PROGRAM _1_LASER
VAR
	FB_LASER_SOURCE_MAXPHOTONICS1: FB_LASER_SOURCE_MAXPHOTONICS;
	FB_LASER_TETE_RAYTOOLS1: FB_LASER_TETE_RAYTOOLS_1;

	Dem_Serrage_Presseur_Entree: BOOL;
	Dem_Desserrage_Presseur_Entree: BOOL;
	Pos_Reelle_Presseur_Entree_D: LREAL;
	Pos_Reelle_Presseur_Entree_G: LREAL;

	Dem_Serrage_Presseur_Sortie: BOOL;
	Dem_Desserrage_Presseur_Sortie: BOOL;
	Pos_Reelle_Presseur_Sortie_D: LREAL;
	Pos_Reelle_Presseur_Sortie_G: LREAL;


	Div_Zero: BOOL;

	Chgt_Plan_Aile_Ref: FB_Calcul_Chgt_Origine_Plan;
	Chgt_Plan_Ame: FB_Calcul_Chgt_Origine_Plan;
	Chgt_Plan_Aile_Opp_Ref: FB_Calcul_Chgt_Origine_Plan;
	
	Feedback_Laser_Power: USINT;
	Feedback_Laser_Duty: USINT;
	Feedback_Laser_Freq: UINT;
	Feedback_Laser_Power_Watts	:UDINT;
	
	
	MeS_Aspiration	:TOF;
	Test_aspi: BOOL;
	Refroidissement	:TOF;
	Test_Refroidissement	:BOOL;
END_VAR
VAR // added by the converter: edge detectors and wires of the graphical bodies
    _w1 : BOOL;
END_VAR

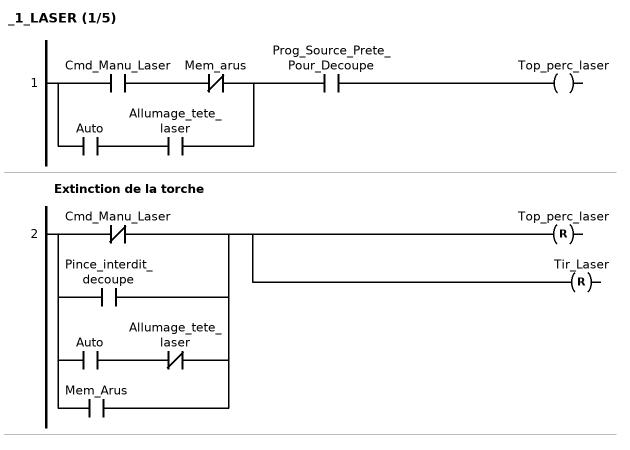
// NETWORK 1
Top_perc_laser := (Cmd_Manu_Laser AND NOT Mem_arus OR Auto AND Allumage_tete_laser) AND Prog_Source_Prete_Pour_Decoupe;

// NETWORK 2: Extinction de la torche
_w1 := NOT Cmd_Manu_Laser OR Pince_interdit_decoupe OR Auto AND NOT Allumage_tete_laser OR Mem_Arus;
Top_perc_laser R= _w1;
Tir_Laser R= _w1;

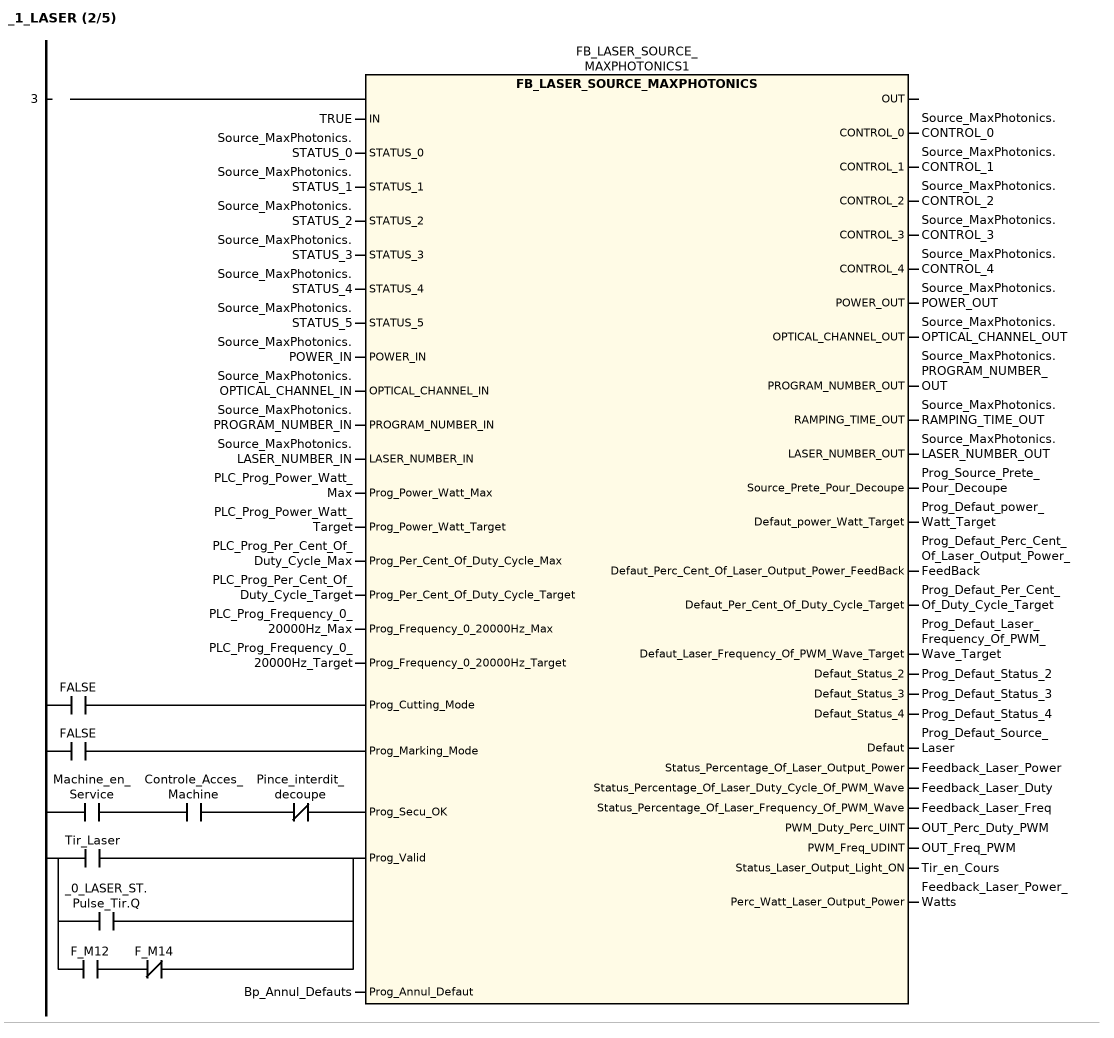
// NETWORK 3
FB_LASER_SOURCE_MAXPHOTONICS1(
    IN := TRUE,
    STATUS_0 := Source_MaxPhotonics.STATUS_0,
    STATUS_1 := Source_MaxPhotonics.STATUS_1,
    STATUS_2 := Source_MaxPhotonics.STATUS_2,
    STATUS_3 := Source_MaxPhotonics.STATUS_3,
    STATUS_4 := Source_MaxPhotonics.STATUS_4,
    STATUS_5 := Source_MaxPhotonics.STATUS_5,
    POWER_IN := Source_MaxPhotonics.POWER_IN,
    OPTICAL_CHANNEL_IN := Source_MaxPhotonics.OPTICAL_CHANNEL_IN,
    PROGRAM_NUMBER_IN := Source_MaxPhotonics.PROGRAM_NUMBER_IN,
    LASER_NUMBER_IN := Source_MaxPhotonics.LASER_NUMBER_IN,
    Prog_Power_Watt_Max := PLC_Prog_Power_Watt_Max,
    Prog_Power_Watt_Target := PLC_Prog_Power_Watt_Target,
    Prog_Per_Cent_Of_Duty_Cycle_Max := PLC_Prog_Per_Cent_Of_Duty_Cycle_Max,
    Prog_Per_Cent_Of_Duty_Cycle_Target := PLC_Prog_Per_Cent_Of_Duty_Cycle_Target,
    Prog_Frequency_0_20000Hz_Max := PLC_Prog_Frequency_0_20000Hz_Max,
    Prog_Frequency_0_20000Hz_Target := PLC_Prog_Frequency_0_20000Hz_Target,
    Prog_Cutting_Mode := FALSE,
    Prog_Marking_Mode := FALSE,
    Prog_Secu_OK := Machine_en_Service AND Controle_Acces_Machine AND NOT Pince_interdit_decoupe,
    Prog_Valid := Tir_Laser OR _0_LASER_ST.Pulse_Tir.Q OR F_M12 AND NOT F_M14,
    Prog_Annul_Defaut := Bp_Annul_Defauts,
    CONTROL_0 => Source_MaxPhotonics.CONTROL_0,
    CONTROL_1 => Source_MaxPhotonics.CONTROL_1,
    CONTROL_2 => Source_MaxPhotonics.CONTROL_2,
    CONTROL_3 => Source_MaxPhotonics.CONTROL_3,
    CONTROL_4 => Source_MaxPhotonics.CONTROL_4,
    POWER_OUT => Source_MaxPhotonics.POWER_OUT,
    OPTICAL_CHANNEL_OUT => Source_MaxPhotonics.OPTICAL_CHANNEL_OUT,
    PROGRAM_NUMBER_OUT => Source_MaxPhotonics.PROGRAM_NUMBER_OUT,
    RAMPING_TIME_OUT => Source_MaxPhotonics.RAMPING_TIME_OUT,
    LASER_NUMBER_OUT => Source_MaxPhotonics.LASER_NUMBER_OUT,
    Source_Prete_Pour_Decoupe => Prog_Source_Prete_Pour_Decoupe,
    Defaut_power_Watt_Target => Prog_Defaut_power_Watt_Target,
    Defaut_Perc_Cent_Of_Laser_Output_Power_FeedBack => Prog_Defaut_Perc_Cent_Of_Laser_Output_Power_FeedBack,
    Defaut_Per_Cent_Of_Duty_Cycle_Target => Prog_Defaut_Per_Cent_Of_Duty_Cycle_Target,
    Defaut_Laser_Frequency_Of_PWM_Wave_Target => Prog_Defaut_Laser_Frequency_Of_PWM_Wave_Target,
    Defaut_Status_2 => Prog_Defaut_Status_2,
    Defaut_Status_3 => Prog_Defaut_Status_3,
    Defaut_Status_4 => Prog_Defaut_Status_4,
    Defaut => Prog_Defaut_Source_Laser,
    Status_Percentage_Of_Laser_Output_Power => Feedback_Laser_Power,
    Status_Percentage_Of_Laser_Duty_Cycle_Of_PWM_Wave => Feedback_Laser_Duty,
    Status_Percentage_Of_Laser_Frequency_Of_PWM_Wave => Feedback_Laser_Freq,
    PWM_Duty_Perc_UINT => OUT_Perc_Duty_PWM,
    PWM_Freq_UDINT => OUT_Freq_PWM,
    Status_Laser_Output_Light_ON => Tir_en_Cours,
    Perc_Watt_Laser_Output_Power => Feedback_Laser_Power_Watts); // FB_LASER_SOURCE_MAXPHOTONICS

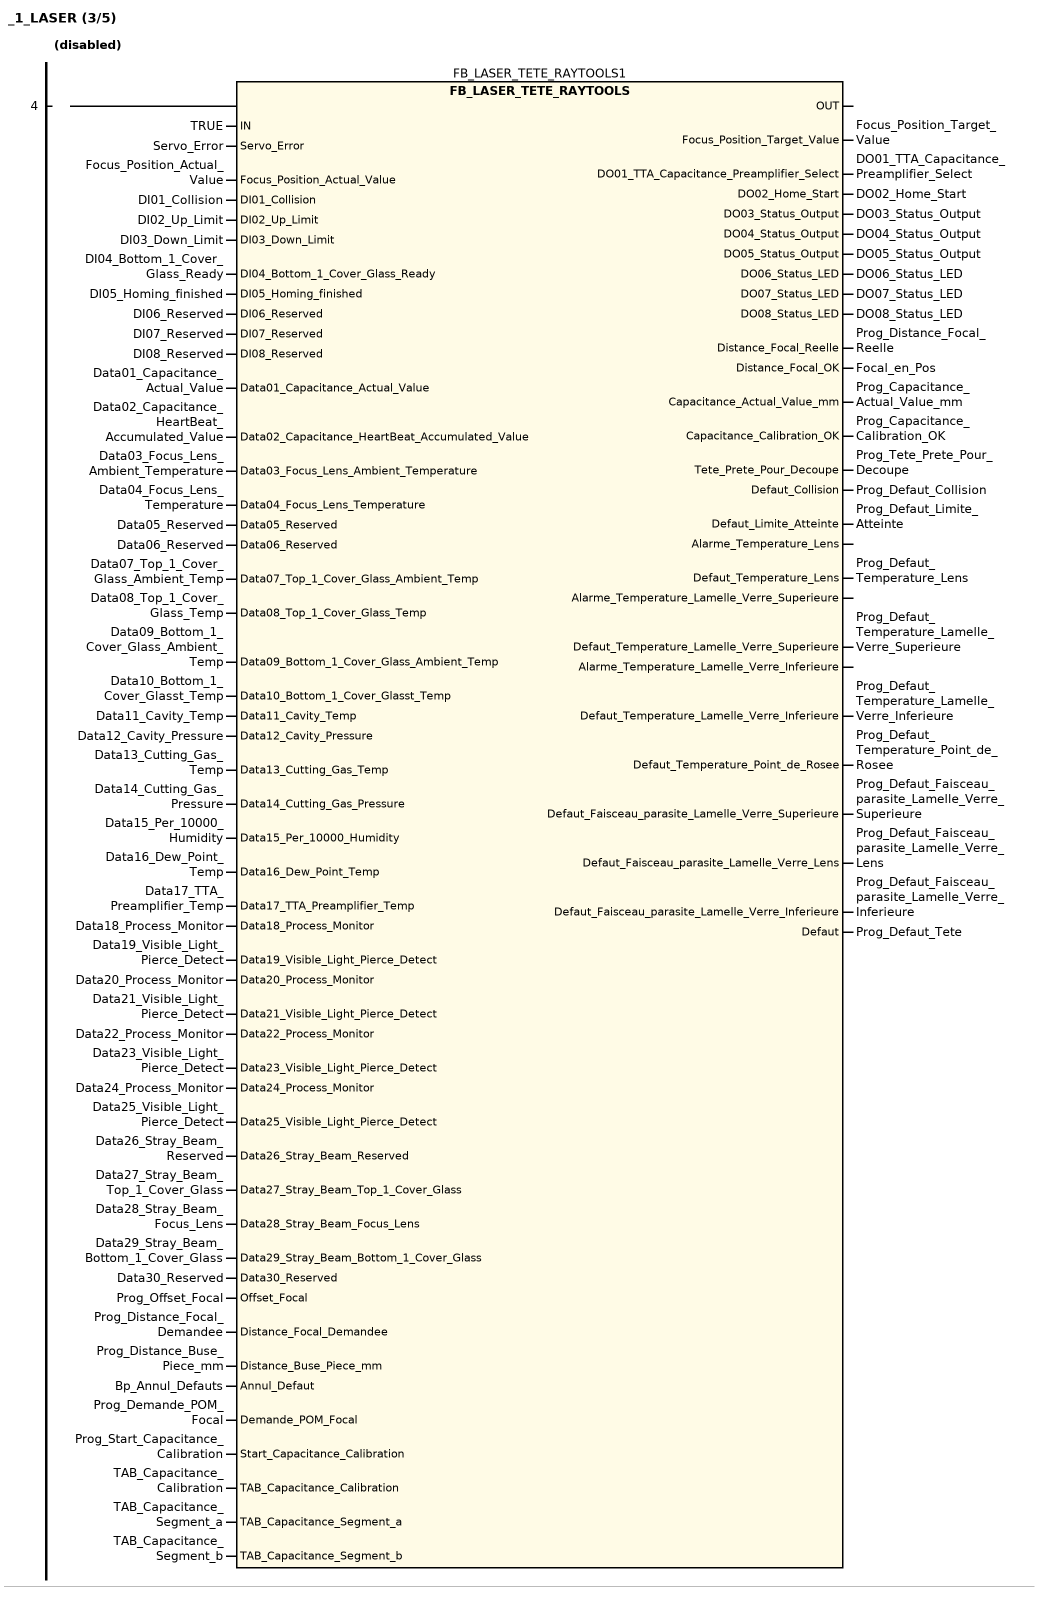
// NETWORK 4 (disabled)
// FB_LASER_TETE_RAYTOOLS1(
//     IN := TRUE,
//     Servo_Error := Servo_Error,
//     Focus_Position_Actual_Value := Focus_Position_Actual_Value,
//     DI01_Collision := DI01_Collision,
//     DI02_Up_Limit := DI02_Up_Limit,
//     DI03_Down_Limit := DI03_Down_Limit,
//     DI04_Bottom_1_Cover_Glass_Ready := DI04_Bottom_1_Cover_Glass_Ready,
//     DI05_Homing_finished := DI05_Homing_finished,
//     DI06_Reserved := DI06_Reserved,
//     DI07_Reserved := DI07_Reserved,
//     DI08_Reserved := DI08_Reserved,
//     Data01_Capacitance_Actual_Value := Data01_Capacitance_Actual_Value,
//     Data02_Capacitance_HeartBeat_Accumulated_Value := Data02_Capacitance_HeartBeat_Accumulated_Value,
//     Data03_Focus_Lens_Ambient_Temperature := Data03_Focus_Lens_Ambient_Temperature,
//     Data04_Focus_Lens_Temperature := Data04_Focus_Lens_Temperature,
//     Data05_Reserved := Data05_Reserved,
//     Data06_Reserved := Data06_Reserved,
//     Data07_Top_1_Cover_Glass_Ambient_Temp := Data07_Top_1_Cover_Glass_Ambient_Temp,
//     Data08_Top_1_Cover_Glass_Temp := Data08_Top_1_Cover_Glass_Temp,
//     Data09_Bottom_1_Cover_Glass_Ambient_Temp := Data09_Bottom_1_Cover_Glass_Ambient_Temp,
//     Data10_Bottom_1_Cover_Glasst_Temp := Data10_Bottom_1_Cover_Glasst_Temp,
//     Data11_Cavity_Temp := Data11_Cavity_Temp,
//     Data12_Cavity_Pressure := Data12_Cavity_Pressure,
//     Data13_Cutting_Gas_Temp := Data13_Cutting_Gas_Temp,
//     Data14_Cutting_Gas_Pressure := Data14_Cutting_Gas_Pressure,
//     Data15_Per_10000_Humidity := Data15_Per_10000_Humidity,
//     Data16_Dew_Point_Temp := Data16_Dew_Point_Temp,
//     Data17_TTA_Preamplifier_Temp := Data17_TTA_Preamplifier_Temp,
//     Data18_Process_Monitor := Data18_Process_Monitor,
//     Data19_Visible_Light_Pierce_Detect := Data19_Visible_Light_Pierce_Detect,
//     Data20_Process_Monitor := Data20_Process_Monitor,
//     Data21_Visible_Light_Pierce_Detect := Data21_Visible_Light_Pierce_Detect,
//     Data22_Process_Monitor := Data22_Process_Monitor,
//     Data23_Visible_Light_Pierce_Detect := Data23_Visible_Light_Pierce_Detect,
//     Data24_Process_Monitor := Data24_Process_Monitor,
//     Data25_Visible_Light_Pierce_Detect := Data25_Visible_Light_Pierce_Detect,
//     Data26_Stray_Beam_Reserved := Data26_Stray_Beam_Reserved,
//     Data27_Stray_Beam_Top_1_Cover_Glass := Data27_Stray_Beam_Top_1_Cover_Glass,
//     Data28_Stray_Beam_Focus_Lens := Data28_Stray_Beam_Focus_Lens,
//     Data29_Stray_Beam_Bottom_1_Cover_Glass := Data29_Stray_Beam_Bottom_1_Cover_Glass,
//     Data30_Reserved := Data30_Reserved,
//     Offset_Focal := Prog_Offset_Focal,
//     Distance_Focal_Demandee := Prog_Distance_Focal_Demandee,
//     Distance_Buse_Piece_mm := Prog_Distance_Buse_Piece_mm,
//     Annul_Defaut := Bp_Annul_Defauts,
//     Demande_POM_Focal := Prog_Demande_POM_Focal,
//     Start_Capacitance_Calibration := Prog_Start_Capacitance_Calibration,
//     TAB_Capacitance_Calibration := TAB_Capacitance_Calibration,
//     TAB_Capacitance_Segment_a := TAB_Capacitance_Segment_a,
//     TAB_Capacitance_Segment_b := TAB_Capacitance_Segment_b,
//     Focus_Position_Target_Value => Focus_Position_Target_Value,
//     DO01_TTA_Capacitance_Preamplifier_Select => DO01_TTA_Capacitance_Preamplifier_Select,
//     DO02_Home_Start => DO02_Home_Start,
//     DO03_Status_Output => DO03_Status_Output,
//     DO04_Status_Output => DO04_Status_Output,
//     DO05_Status_Output => DO05_Status_Output,
//     DO06_Status_LED => DO06_Status_LED,
//     DO07_Status_LED => DO07_Status_LED,
//     DO08_Status_LED => DO08_Status_LED,
//     Distance_Focal_Reelle => Prog_Distance_Focal_Reelle,
//     Distance_Focal_OK => Focal_en_Pos,
//     Capacitance_Actual_Value_mm => Prog_Capacitance_Actual_Value_mm,
//     Capacitance_Calibration_OK => Prog_Capacitance_Calibration_OK,
//     Tete_Prete_Pour_Decoupe => Prog_Tete_Prete_Pour_Decoupe,
//     Defaut_Collision => Prog_Defaut_Collision,
//     Defaut_Limite_Atteinte => Prog_Defaut_Limite_Atteinte,
//     Defaut_Temperature_Lens => Prog_Defaut_Temperature_Lens,
//     Defaut_Temperature_Lamelle_Verre_Superieure => Prog_Defaut_Temperature_Lamelle_Verre_Superieure,
//     Defaut_Temperature_Lamelle_Verre_Inferieure => Prog_Defaut_Temperature_Lamelle_Verre_Inferieure,
//     Defaut_Temperature_Point_de_Rosee => Prog_Defaut_Temperature_Point_de_Rosee,
//     Defaut_Faisceau_parasite_Lamelle_Verre_Superieure => Prog_Defaut_Faisceau_parasite_Lamelle_Verre_Superieure,
//     Defaut_Faisceau_parasite_Lamelle_Verre_Lens => Prog_Defaut_Faisceau_parasite_Lamelle_Verre_Lens,
//     Defaut_Faisceau_parasite_Lamelle_Verre_Inferieure => Prog_Defaut_Faisceau_parasite_Lamelle_Verre_Inferieure,
//     Defaut => Prog_Defaut_Tete); // FB_LASER_TETE_RAYTOOLS

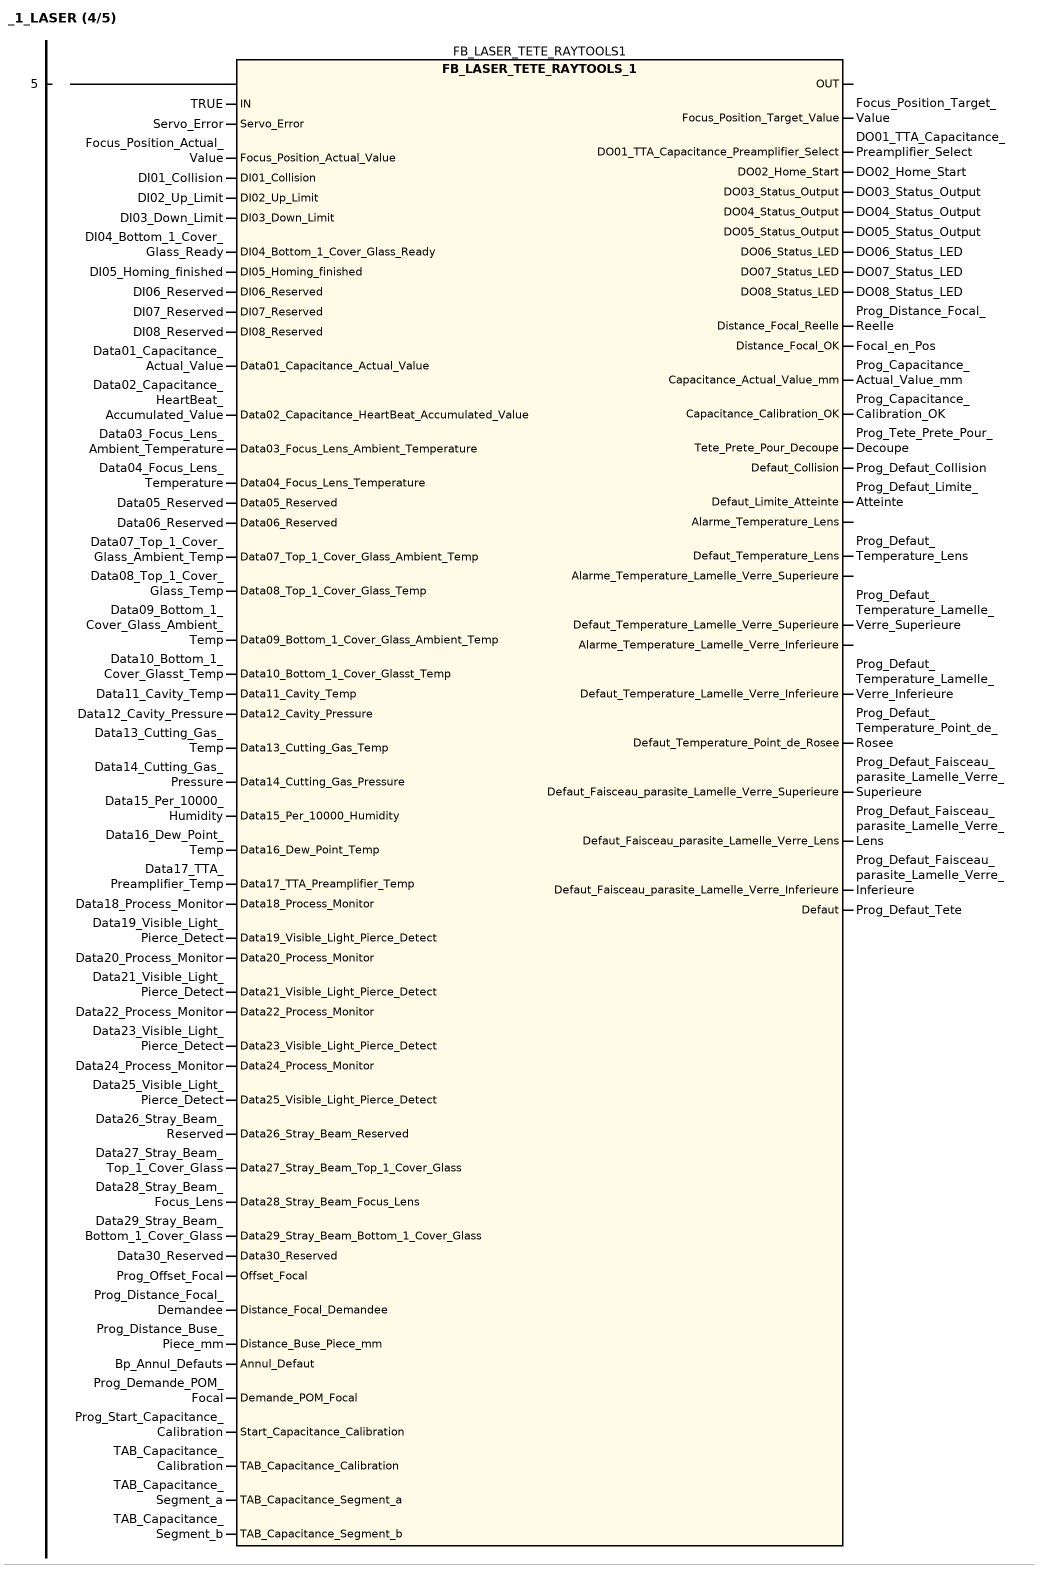
// NETWORK 5
FB_LASER_TETE_RAYTOOLS1(
    IN := TRUE,
    Servo_Error := Servo_Error,
    Focus_Position_Actual_Value := Focus_Position_Actual_Value,
    DI01_Collision := DI01_Collision,
    DI02_Up_Limit := DI02_Up_Limit,
    DI03_Down_Limit := DI03_Down_Limit,
    DI04_Bottom_1_Cover_Glass_Ready := DI04_Bottom_1_Cover_Glass_Ready,
    DI05_Homing_finished := DI05_Homing_finished,
    DI06_Reserved := DI06_Reserved,
    DI07_Reserved := DI07_Reserved,
    DI08_Reserved := DI08_Reserved,
    Data01_Capacitance_Actual_Value := Data01_Capacitance_Actual_Value,
    Data02_Capacitance_HeartBeat_Accumulated_Value := Data02_Capacitance_HeartBeat_Accumulated_Value,
    Data03_Focus_Lens_Ambient_Temperature := Data03_Focus_Lens_Ambient_Temperature,
    Data04_Focus_Lens_Temperature := Data04_Focus_Lens_Temperature,
    Data05_Reserved := Data05_Reserved,
    Data06_Reserved := Data06_Reserved,
    Data07_Top_1_Cover_Glass_Ambient_Temp := Data07_Top_1_Cover_Glass_Ambient_Temp,
    Data08_Top_1_Cover_Glass_Temp := Data08_Top_1_Cover_Glass_Temp,
    Data09_Bottom_1_Cover_Glass_Ambient_Temp := Data09_Bottom_1_Cover_Glass_Ambient_Temp,
    Data10_Bottom_1_Cover_Glasst_Temp := Data10_Bottom_1_Cover_Glasst_Temp,
    Data11_Cavity_Temp := Data11_Cavity_Temp,
    Data12_Cavity_Pressure := Data12_Cavity_Pressure,
    Data13_Cutting_Gas_Temp := Data13_Cutting_Gas_Temp,
    Data14_Cutting_Gas_Pressure := Data14_Cutting_Gas_Pressure,
    Data15_Per_10000_Humidity := Data15_Per_10000_Humidity,
    Data16_Dew_Point_Temp := Data16_Dew_Point_Temp,
    Data17_TTA_Preamplifier_Temp := Data17_TTA_Preamplifier_Temp,
    Data18_Process_Monitor := Data18_Process_Monitor,
    Data19_Visible_Light_Pierce_Detect := Data19_Visible_Light_Pierce_Detect,
    Data20_Process_Monitor := Data20_Process_Monitor,
    Data21_Visible_Light_Pierce_Detect := Data21_Visible_Light_Pierce_Detect,
    Data22_Process_Monitor := Data22_Process_Monitor,
    Data23_Visible_Light_Pierce_Detect := Data23_Visible_Light_Pierce_Detect,
    Data24_Process_Monitor := Data24_Process_Monitor,
    Data25_Visible_Light_Pierce_Detect := Data25_Visible_Light_Pierce_Detect,
    Data26_Stray_Beam_Reserved := Data26_Stray_Beam_Reserved,
    Data27_Stray_Beam_Top_1_Cover_Glass := Data27_Stray_Beam_Top_1_Cover_Glass,
    Data28_Stray_Beam_Focus_Lens := Data28_Stray_Beam_Focus_Lens,
    Data29_Stray_Beam_Bottom_1_Cover_Glass := Data29_Stray_Beam_Bottom_1_Cover_Glass,
    Data30_Reserved := Data30_Reserved,
    Offset_Focal := Prog_Offset_Focal,
    Distance_Focal_Demandee := Prog_Distance_Focal_Demandee,
    Distance_Buse_Piece_mm := Prog_Distance_Buse_Piece_mm,
    Annul_Defaut := Bp_Annul_Defauts,
    Demande_POM_Focal := Prog_Demande_POM_Focal,
    Start_Capacitance_Calibration := Prog_Start_Capacitance_Calibration,
    TAB_Capacitance_Calibration := TAB_Capacitance_Calibration,
    TAB_Capacitance_Segment_a := TAB_Capacitance_Segment_a,
    TAB_Capacitance_Segment_b := TAB_Capacitance_Segment_b,
    Focus_Position_Target_Value => Focus_Position_Target_Value,
    DO01_TTA_Capacitance_Preamplifier_Select => DO01_TTA_Capacitance_Preamplifier_Select,
    DO02_Home_Start => DO02_Home_Start,
    DO03_Status_Output => DO03_Status_Output,
    DO04_Status_Output => DO04_Status_Output,
    DO05_Status_Output => DO05_Status_Output,
    DO06_Status_LED => DO06_Status_LED,
    DO07_Status_LED => DO07_Status_LED,
    DO08_Status_LED => DO08_Status_LED,
    Distance_Focal_Reelle => Prog_Distance_Focal_Reelle,
    Distance_Focal_OK => Focal_en_Pos,
    Capacitance_Actual_Value_mm => Prog_Capacitance_Actual_Value_mm,
    Capacitance_Calibration_OK => Prog_Capacitance_Calibration_OK,
    Tete_Prete_Pour_Decoupe => Prog_Tete_Prete_Pour_Decoupe,
    Defaut_Collision => Prog_Defaut_Collision,
    Defaut_Limite_Atteinte => Prog_Defaut_Limite_Atteinte,
    Defaut_Temperature_Lens => Prog_Defaut_Temperature_Lens,
    Defaut_Temperature_Lamelle_Verre_Superieure => Prog_Defaut_Temperature_Lamelle_Verre_Superieure,
    Defaut_Temperature_Lamelle_Verre_Inferieure => Prog_Defaut_Temperature_Lamelle_Verre_Inferieure,
    Defaut_Temperature_Point_de_Rosee => Prog_Defaut_Temperature_Point_de_Rosee,
    Defaut_Faisceau_parasite_Lamelle_Verre_Superieure => Prog_Defaut_Faisceau_parasite_Lamelle_Verre_Superieure,
    Defaut_Faisceau_parasite_Lamelle_Verre_Lens => Prog_Defaut_Faisceau_parasite_Lamelle_Verre_Lens,
    Defaut_Faisceau_parasite_Lamelle_Verre_Inferieure => Prog_Defaut_Faisceau_parasite_Lamelle_Verre_Inferieure,
    Defaut => Prog_Defaut_Tete); // FB_LASER_TETE_RAYTOOLS_1

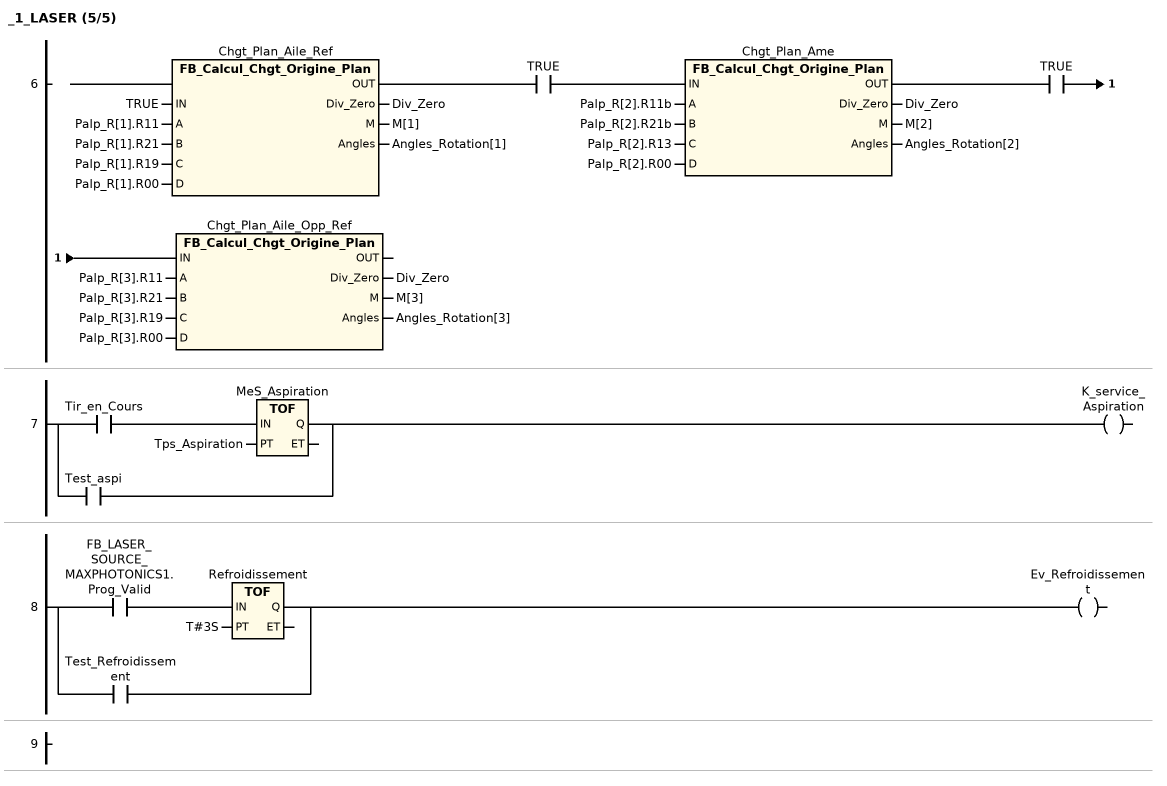
// NETWORK 6
Chgt_Plan_Aile_Ref(
    IN := TRUE,
    A := Palp_R[1].R11,
    B := Palp_R[1].R21,
    C := Palp_R[1].R19,
    D := Palp_R[1].R00,
    Div_Zero => Div_Zero,
    M => M[1],
    Angles => Angles_Rotation[1]); // FB_Calcul_Chgt_Origine_Plan
Chgt_Plan_Ame(
    IN := Chgt_Plan_Aile_Ref.OUT AND TRUE,
    A := Palp_R[2].R11b,
    B := Palp_R[2].R21b,
    C := Palp_R[2].R13,
    D := Palp_R[2].R00,
    Div_Zero => Div_Zero,
    M => M[2],
    Angles => Angles_Rotation[2]); // FB_Calcul_Chgt_Origine_Plan
Chgt_Plan_Aile_Opp_Ref(
    IN := Chgt_Plan_Ame.OUT AND TRUE,
    A := Palp_R[3].R11,
    B := Palp_R[3].R21,
    C := Palp_R[3].R19,
    D := Palp_R[3].R00,
    Div_Zero => Div_Zero,
    M => M[3],
    Angles => Angles_Rotation[3]); // FB_Calcul_Chgt_Origine_Plan

// NETWORK 7
MeS_Aspiration(IN := Tir_en_Cours, PT := Tps_Aspiration); // TOF
K_service_Aspiration := MeS_Aspiration.Q OR Test_aspi;

// NETWORK 8
Refroidissement(IN := FB_LASER_SOURCE_MAXPHOTONICS1.Prog_Valid, PT := T#3S); // TOF
Ev_Refroidissement := Refroidissement.Q OR Test_Refroidissement;

// NETWORK 9

END_PROGRAM

(* stored: Version 1.1.0.1
   POU _1_LASER: Id {5ec5b7da-aae7-40d7-a08e-c40004e74d06}, SpecialFunc None *)
